FUNCTION_BLOCK automatic
VAR_INPUT
	LDR1, LDR2		: INT;
	LDR_threshold	: INT;
	LDR_duty		: INT;
	motion			: BOOL;
END_VAR
VAR_OUTPUT
	fQ	: BOOL;
	rQ	: BOOL;
END_VAR
VAR
	Motion_ton	: TON;
	Motion_tof	: TOF;
	LDR_tof		: TOF;
	fTRIG: F_TRIG;
	rTRIG: R_TRIG;
	LDR_low: BOOL;
	hys1: hysterisis;
	hys2: hysterisis;
END_VAR

Motion_ton( IN := motion, PT := T#1S );
Motion_tof( IN := Motion_ton.Q, PT := T#5M );

hys1(IN:= LDR1, thresh:= LDR_threshold, variatie:= LDR_duty );
hys2(IN:= LDR2, thresh:= LDR_threshold, variatie:= LDR_duty );

IF Motion_tof.Q THEN
	IF (hys1.UP) AND NOT(hys2.UP) ) THEN
	IF (LDR1 < LDR_threshold) OR (LDR2 < LDR_threshold) THEN
		LDR_low := TRUE;
	ELSIF (LDR1 > LDR_threshold) OR (LDR2 < LDR_threshold)
		LDR_tof.IN := FALSE;
	END_IF
ELSE
	LDR_tof.IN := FALSE;
END_IF

LDR_tof( PT := T#1M );

fTRIG(CLK := LDR_tof.Q ,Q=> );
rTRIG(CLK := LDR_tof.Q ,Q=> );

END_FUNCTION_BLOCK

(* stored: Version 1.1.0.1, ProductVersion 3.1.4022.12
   POU automatic: Id {42be8525-c00d-4368-b96c-2cea286f2f01}, SpecialFunc None *)
